(*udt (user defined type) of Beckhoff EL2622 - 2 Point Relay Type Output Terminal:
	auth. Brent Lekx-Toniolo of Toniolo Research & Development Inc.; 
	July 2010; version 1.0*)


TYPE udt_EL2622 :
STRUCT
	Q0: BOOL;
	Q1: BOOL;
END_STRUCT
END_TYPE

(* stored: Version 1.1.0.1, ProductVersion 3.1.4024.9
   DUT udt_EL2622: Id {b41d2363-2865-443b-851b-55c232670148} *)
